// TwinCAT 3 PLC project Sample_Delivery
// ProgramVersion: 3.1.4023.0
// libraries:
//   LCLS General, * (SLAC)
//   LCLS Vacuum, * (SLAC - LCLS)
//   Tc2_Standard, * (Beckhoff Automation GmbH)
//   Tc2_System, * (Beckhoff Automation GmbH)
//   Tc3_Module, * (Beckhoff Automation GmbH)
// project tree:
//   GVLs/ GVL_RCC.TcGVL (not stored)
//   / PlcTask.TcTTO (not stored)
//   POUs/ FB_RCC_Valves.TcPOU, MAIN.TcPOU, PRG_RCC.TcPOU
// real-time tasks:
//   TASK PlcTask: cycle T#10ms, priority 20, ADS port 350
// I/O:
//   DEVICE Device 1 (EtherCAT), AmsNetId 172.21.148.84.2.1
//     Term 4 (EK1200) [EK1200-5000 EtherCAT Power supply (2A E-Bus)]
//       RCC_E1 (EL2004) [EL2004 4Ch. Dig. Output 24V, 0.5A]
//       RCC_E2 (EL1004) [EL1004 4Ch. Dig. Input 24V, 3ms]
//       RCC_E3 (EL1004) [EL1004 4Ch. Dig. Input 24V, 3ms]
//       RCC_TC (EL3314) [EL3314 4Ch. Ana. Input Thermocouple (TC)]
//       Term 9 (EK1110) [EK1110 EtherCAT extension]
// variable links:
//   Sample_Delivery Instance <-> Device 1 (EtherCAT)/Term 1 (EK1200)/RCC_E1 (EL2004)
//     PlcTask Outputs/GVL_RCC.RCC_VRC_01.q_xOPN_DO <-> Channel 1/Output
//     PlcTask Outputs/GVL_RCC.RCC_VRC_02.q_xOPN_DO <-> Channel 2/Output
//     PlcTask Outputs/GVL_RCC.RCC_VRC_03.q_xOPN_DO <-> Channel 3/Output
//     PlcTask Outputs/GVL_RCC.RCC_VRC_04.q_xOPN_DO <-> Channel 4/Output
//   Sample_Delivery Instance <-> Device 1 (EtherCAT)/Term 1 (EK1200)/RCC_E2 (EL1004)
//     PlcTask Inputs/GVL_RCC.RCC_VRC_01.i_xClsLS <-> Channel 1/Input
//     PlcTask Inputs/GVL_RCC.RCC_VRC_02.i_xClsLS <-> Channel 4/Input
//     PlcTask Inputs/GVL_RCC.RCC_VRC_02.i_xOpnLS <-> Channel 3/Input
//   Sample_Delivery Instance <-> Device 1 (EtherCAT)/Term 1 (EK1200)/RCC_E3 (EL1004)
//     PlcTask Inputs/GVL_RCC.RCC_VRC_03.i_xClsLS <-> Channel 1/Input
//     PlcTask Inputs/GVL_RCC.RCC_VRC_04.i_xClsLS <-> Channel 1/Input
//   Sample_Delivery Instance <-> Device 1 (EtherCAT)/Term 1 (EK1200)/RCC_TC (EL3314)
//     PlcTask Inputs/GVL_RCC.RCC_STC_01.bError <-> TC Inputs Channel 1/Status/Error
//     PlcTask Inputs/GVL_RCC.RCC_STC_01.bOverrange <-> TC Inputs Channel 1/Status/Overrange
//     PlcTask Inputs/GVL_RCC.RCC_STC_01.bUnderrange <-> TC Inputs Channel 1/Status/Underrange
//     PlcTask Inputs/GVL_RCC.RCC_STC_01.iRaw <-> TC Inputs Channel 1/Value

// ---- POUs/FB_RCC_Valves.TcPOU
FUNCTION_BLOCK FB_RCC_Valves
VAR_INPUT
      RCC_VRC_01 : FB_VRC_NC_ClsLS;
      RCC_VRC_02 : FB_VRC;
      RCC_VRC_03 : FB_VRC_NC_ClsLS;
      RCC_VRC_04 : FB_VRC_NC_ClsLS;

      RCC_GCP_01 : FB_901_ECAT;
      RCC_GCP_01_INTERLOCK_SETPOINT : REAL;
END_VAR
VAR
    RCC_VRC_01_OPEN_OK : BOOL;
    RCC_VRC_02_OPEN_OK : BOOL;
    RCC_VRC_03_OPEN_OK : BOOL;
    RCC_VRC_04_OPEN_OK : BOOL;
END_VAR

RCC_GCP_01(PG=>);

(* Valve can open only when RCC-VRC-02 and 03 are closed*)
RCC_VRC_01_OPEN_OK := ( RCC_VRC_02.iq_stValve.i_xClsLS AND NOT RCC_VRC_02.iq_stValve.q_xOPN_DO ) AND
                                    ( RCC_VRC_03.iq_stValve.i_xClsLS AND NOT RCC_VRC_03.iq_stValve.q_xOPN_DO ) ;

RCC_VRC_01(i_xExtILK_OK := RCC_VRC_01_OPEN_OK,
                i_xOverrideMode := xSystemOverrideMode_RCC,
                 iq_stValve=> );

(* Valve can open only when RCC-VRC-01 and 04 are closed*)
RCC_VRC_02_OPEN_OK := ( RCC_VRC_01.iq_stValve.i_xClsLS AND NOT RCC_VRC_01.iq_stValve.q_xOPN_DO ) AND
                                    ( RCC_VRC_04.iq_stValve.i_xClsLS AND NOT RCC_VRC_04.iq_stValve.q_xOPN_DO );

RCC_VRC_02(i_xExtILK_OK := RCC_VRC_02_OPEN_OK,
                i_xOverrideMode := xSystemOverrideMode_RCC,
                 iq_stValve=> );

(* Valve can open only when RCC-GCP-01 reading < setpoint Torr and RCC-VRC-01 and 04 are closed*)
RCC_VRC_03_OPEN_OK := (RCC_GCP_01.PG.rPRESS < RCC_GCP_01_INTERLOCK_SETPOINT and RCC_GCP_01.PG.xPRESS_OK ) AND
                                 ( RCC_VRC_01.iq_stValve.i_xClsLS AND NOT RCC_VRC_01.iq_stValve.q_xOPN_DO ) AND
                                              ( RCC_VRC_04.iq_stValve.i_xClsLS AND NOT RCC_VRC_04.iq_stValve.q_xOPN_DO );

RCC_VRC_03(i_xExtILK_OK := RCC_VRC_03_OPEN_OK,
                i_xOverrideMode := xSystemOverrideMode_RCC,
                 iq_stValve=> );

(* Valve can open only when RCC-VRC-02 and 03 are closed*)
RCC_VRC_04_OPEN_OK := ( RCC_VRC_02.iq_stValve.i_xClsLS AND NOT RCC_VRC_02.iq_stValve.q_xOPN_DO ) AND
                                      ( RCC_VRC_03.iq_stValve.i_xClsLS AND NOT RCC_VRC_03.iq_stValve.q_xOPN_DO ) ;

RCC_VRC_04(i_xExtILK_OK := RCC_VRC_04_OPEN_OK,
                i_xOverrideMode := xSystemOverrideMode_RCC,
                 iq_stValve=> );

END_FUNCTION_BLOCK

// ---- POUs/MAIN.TcPOU
PROGRAM MAIN
VAR
END_VAR

//PRG_RCC();

END_PROGRAM

// ---- POUs/PRG_RCC.TcPOU
PROGRAM PRG_RCC
VAR
    RCC_VRC_01_OPEN_OK : BOOL;
    RCC_VRC_02_OPEN_OK : BOOL;
    RCC_VRC_03_OPEN_OK : BOOL;
    RCC_VRC_04_OPEN_OK : BOOL;

   {attribute 'pytmc' :=' pv: UED:GCP:01:INLK_Setpoint '}
    RCC_GCP_01_INTERLOCK_SETPOINT : REAL := 10;

END_VAR

RCC_GCP_01(PG=>);
RCC_STC_01();

(* Valve can open only when UED-RCC-VRC-02 and 03 are closed*)
RCC_VRC_01_OPEN_OK := ( RCC_VRC_02.iq_stValve.i_xClsLS AND NOT RCC_VRC_02.iq_stValve.q_xOPN_DO ) AND
                                    ( RCC_VRC_03.iq_stValve.i_xClsLS AND NOT RCC_VRC_03.iq_stValve.q_xOPN_DO ) ;

RCC_VRC_01(i_xExtILK_OK := RCC_VRC_01_OPEN_OK,
                i_xOverrideMode := xSystemOverrideMode_RCC,
                 iq_stValve=> );

(* Valve can open only when UED-RCC-VRC-01 and 04 are closed*)
RCC_VRC_02_OPEN_OK := ( RCC_VRC_01.iq_stValve.i_xClsLS AND NOT RCC_VRC_01.iq_stValve.q_xOPN_DO ) AND
                                    ( RCC_VRC_04.iq_stValve.i_xClsLS AND NOT RCC_VRC_04.iq_stValve.q_xOPN_DO );

RCC_VRC_02(i_xExtILK_OK := RCC_VRC_02_OPEN_OK,
                i_xOverrideMode := xSystemOverrideMode_RCC,
                 iq_stValve=> );

(* Valve can open only when UED-RCC-GCP-01 reading < setpoint Torr and UED-RCC-VRC-01 and 04 are closed*)
RCC_VRC_03_OPEN_OK := (RCC_GCP_01.PG.rPRESS < RCC_GCP_01_INTERLOCK_SETPOINT and RCC_GCP_01.PG.xPRESS_OK ) AND
                                 ( RCC_VRC_01.iq_stValve.i_xClsLS AND NOT RCC_VRC_01.iq_stValve.q_xOPN_DO ) AND
                                              ( RCC_VRC_04.iq_stValve.i_xClsLS AND NOT RCC_VRC_04.iq_stValve.q_xOPN_DO );

RCC_VRC_03(i_xExtILK_OK := RCC_VRC_03_OPEN_OK,
                i_xOverrideMode := xSystemOverrideMode_RCC,
                 iq_stValve=> );

(* Valve can open only when UED-RCC-VRC-02 and 03 are closed*)
RCC_VRC_04_OPEN_OK := ( RCC_VRC_02.iq_stValve.i_xClsLS AND NOT RCC_VRC_02.iq_stValve.q_xOPN_DO ) AND
                                      ( RCC_VRC_03.iq_stValve.i_xClsLS AND NOT RCC_VRC_03.iq_stValve.q_xOPN_DO ) ;

RCC_VRC_04(i_xExtILK_OK := RCC_VRC_04_OPEN_OK,
                i_xOverrideMode := xSystemOverrideMode_RCC,
                 iq_stValve=> );

END_PROGRAM
